PROGRAM INTERNAL PRG_TESTS

(* Instantiate test suites here. Naming convention for tests should be a suffix with _Tests.
Good practice for creating test methods is to end them with _test as well. *)
VAR
	LightTowerComponentTest	: FB_LightTowerComponent_Tests;
	FqInverter_IOTests		: FB_FqInverter_IO_Tests;
	LighttowerTests			: FB_LightTower_Tests;
END_VAR

// Run tests in paralel
//TcUnit.RUN();

// Run tests in sequence, one after the other. Uncomment if required.
TcUnit.RUN_IN_SEQUENCE();

END_PROGRAM

(* stored: Version 1.1.0.1, ProductVersion 3.1.4024.16
   POU PRG_TESTS: Id {1113ab77-bf03-4669-9da6-9a0d4175f9c5}, SpecialFunc None *)
